// TIA Portal project "Simulador_De_Tren" (V19)

(* hardware
DEVICE "S7-1500/ET200MP station_1"  S7-1500 station
   slot 0: "Rail_0"  Rack  6ES7 590-1***0-0AA0
   slot 1: "PLC_1"  CPU 1511-1 PN  6ES7 511-1AK01-0AB0  V2.9
      slot 3: "CPU display_1"  6ES7591-1AA00-0AA0
      slot 32768: "PROFINET interface_1"  X1
         slot 32769: "Port_1"  X1 P1
         slot 32770: "Port_2"  X1 P2
      slot 34817: "Virtual CP interface port_1"  Virtual CP interface port  Virtual CP interface port
   slot 2: "DI 32x24VDC BA_1"  DI 32x24VDC BA  6ES7 521-1BL10-0AA0  V1.1
   slot 3: "DQ 32x24VDC/0.5A BA_1"  DQ 32x24VDC/0.5A BA  6ES7 522-1BL10-0AA0  V1.1
   slot 4: "AI 16xI BA_1"  AI 16xI BA  6ES7 531-7MH00-0AB0  V1.0
   slot 5: "AQ 8xU/I HS_1"  AQ 8xU/I HS  6ES7 532-5HF00-0AB0  V2.2
DEVICE "HMI_1"  TP1500 Comfort
   slot 0: "HMI_1"  TP1500 Comfort  6AV2 124-0QC02-0AX1  17.0.0.0
   slot 1: "HMI_RT_1"  TP1500 Comfort  6AV2 124-0QC02-0AX1  17.0.0.0
   slot 5: "HMI_1.IE_CP_1"  PROFINET Interface  17.0.0.0
      slot 1: "PROFINET Interface_1"  PROFINET Interface
         slot 1: "Port_1"  Port
         slot 2: "Port_2"  Port
   slot 6: "HMI_1.IE_CP_2"  PROFINET Interface  17.0.0.0
      slot 1: "PROFINET Interface_GBit"  PROFINET Interface
         slot 1: "Port_1"  Port
   slot 7: "HMI_1.MPI/DP_CP_1"  MPI/DP Interface  17.0.0.0
*)

// ===== PLC "PLC_1"  CPU 1511-1 PN =====

VAR_GLOBAL   // PLC tag table "Default tag table"
   "VT-01_TrainVibration" AT %IW4 : Int;
   "M-01-SPD_Mtr1Speed" AT %QW4 : Int;
END_VAR

VAR_GLOBAL   // PLC tag table "DigitalInputs"
   "ZS-01_LowLevel" AT %I0.0 : Bool;
   "ZS-02_HighLeve" AT %I0.1 : Bool;
   "ZS-03_MediumLevel" AT %I0.2 : Bool;
   "ZS-04" AT %I0.3 : Bool;
   "ZS-05" AT %I0.4 : Bool;
   "ZS-06" AT %I0.5 : Bool;
   "ZS-07" AT %I0.6 : Bool;
   "ZS-08" AT %I0.7 : Bool;
END_VAR

VAR_GLOBAL   // PLC tag table "DigitalOutputs"
   "M-01-Run_Mtr1RunCmd" AT %Q0.0 : Bool;
END_VAR

DATA_BLOCK "M-01"   // DB7
{ S7_Optimized_Access := 'TRUE' }
VERSION : 0.1
// stored: InstanceOfName FB_Motor_VSD
"FB_Motor_VSD"
BEGIN
END_DATA_BLOCK

DATA_BLOCK "M-02"   // DB8
{ S7_Optimized_Access := 'TRUE' }
VERSION : 0.1
// stored: InstanceOfName FB_Motor_VSD
"FB_Motor_VSD"
BEGIN
END_DATA_BLOCK

// folder: 1.IO_DB's

DATA_BLOCK "DI"   // DB1
{ S7_Optimized_Access := 'TRUE' }
VERSION : 0.1
   VAR
      "ZS-01_Fault_Rev" : Bool;
      "ZS-02_Stop1" : Bool;
      "ZS-03_Slow1_Rev" : Bool;
      "ZS-04_Slow2_Fwd" : Bool;
      "ZS-05_Stop2" : Bool;
      "ZS-06_Slow2_Rev" : Bool;
      "ZS-07_Slow3_Fwd" : Bool;
      "ZS-08_Stop3" : Bool;
      "ZS-09_Slow3_Rev" : Bool;
      "ZS-10_Slow4_Fwd" : Bool;
      "ZS-11_Stop4" : Bool;
      "ZS-12_Fault_Fwd" : Bool;
      "!XS--01_E-Stop" : Bool;
      "!XS-02_Safety_Key" : Bool;
      "!LS-01_LIght_Curtain" : Bool;
      "M-01-Ctrl_Flt" : Bool;
      "M-01-VSD_Flt" : Bool;
      "ZS-13_Brake_Engaged" : Bool;
      "M-01-Run_Conf" : Bool;
   END_VAR
BEGIN
END_DATA_BLOCK

DATA_BLOCK "DO"   // DB2
{ S7_Optimized_Access := 'TRUE' }
VERSION : 0.1
   VAR
      "XZ-01_Brake_Cmd" : Bool;
      "M-01_Run_Cmd" : Bool;
      "M-01_Mtr_Dir_Fwd" : Bool;
   END_VAR
BEGIN
END_DATA_BLOCK

DATA_BLOCK "AI"   // DB3
{ S7_Optimized_Access := 'TRUE' }
VERSION : 0.1
   VAR
      "VT-01_Train_Vibration" : Int;
   END_VAR
BEGIN
END_DATA_BLOCK

DATA_BLOCK "AO"   // DB4
{ S7_Optimized_Access := 'TRUE' }
VERSION : 0.1
   VAR
      "M-01_Mtr_Spd" : Int;
      "M-01_Mtr_Accl" : Int;
   END_VAR
BEGIN
END_DATA_BLOCK

DATA_BLOCK "HMI_Inputs"   // DB5
{ S7_Optimized_Access := 'TRUE' }
VERSION : 0.1
   VAR
      GoTo_Station1 : Bool;
      GoTo_Station2 : Bool;
      GoTo_Station3 : Bool;
      GoTo_Station4 : Bool;
   END_VAR
BEGIN
END_DATA_BLOCK

DATA_BLOCK "Const&SP"   // DB6
{ S7_Optimized_Access := 'TRUE' }
VERSION : 0.1
BEGIN
END_DATA_BLOCK

DATA_BLOCK "TestDB"   // DB9
{ S7_Optimized_Access := 'TRUE' }
VERSION : 0.1
   VAR
      Test_faultVSD : Bool;
      Test_Start : Bool;
      Test_Stop : Bool;
      Test_FWD : Bool;
      Test_Reset : Bool;
   END_VAR
BEGIN
END_DATA_BLOCK

// folder: (top level)

ORGANIZATION_BLOCK "Main"   // OB1, LAD, ProgramCycle
TITLE = "Main Program Sweep (Cycle)"
{ S7_Optimized_Access := 'TRUE' }
VERSION : 0.1
   VAR_INPUT
      Initial_Call : Bool;   // Initial call of this OB
      Remanence : Bool;   // =True, if remanent data are available
   END_VAR
BEGIN

REGION Network 1
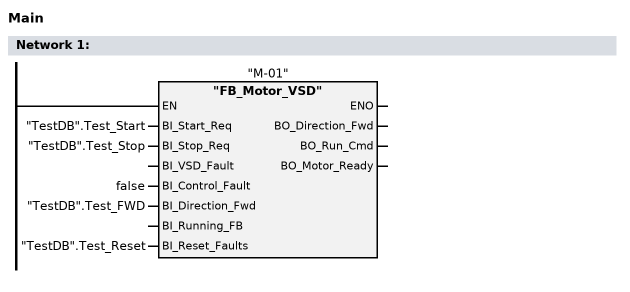
   RUNG wire#powerrail
      "M-01"(BI_Start_Req := "TestDB".Test_Start, BI_Stop_Req := "TestDB".Test_Stop, BI_VSD_Fault :=, BI_Control_Fault := false, BI_Direction_Fwd := "TestDB".Test_FWD, BI_Running_FB :=, BI_Reset_Faults := "TestDB".Test_Reset, BO_Direction_Fwd =>, BO_Run_Cmd =>, BO_Motor_Ready =>)
   END_RUNG
   // the same network as SCL:
   "M-01"(BI_Start_Req := "TestDB".Test_Start,   // "FB_Motor_VSD"
          BI_Stop_Req := "TestDB".Test_Stop,
          BI_Control_Fault := false,
          BI_Direction_Fwd := "TestDB".Test_FWD,
          BI_Reset_Faults := "TestDB".Test_Reset);
END_REGION
END_ORGANIZATION_BLOCK

// folder: 2.Function_Blocks

FUNCTION_BLOCK "FB_Motor_VSD"   // FB1, LAD
TITLE = Function block for control of a VSD Motor
{ S7_Optimized_Access := 'TRUE' }
VERSION : 0.1
   VAR_INPUT
      BI_Start_Req : Bool;
      BI_Stop_Req : Bool;
      BI_VSD_Fault : Bool;
      BI_Control_Fault : Bool;
      BI_Direction_Fwd : Bool;
      BI_Running_FB : Bool;
      BI_Reset_Faults : Bool;
   END_VAR
   VAR_OUTPUT
      BO_Direction_Fwd : Bool;
      BO_Run_Cmd : Bool;
      BO_Motor_Ready : Bool;
      BO_Running_Sts : Bool;
   END_VAR
BEGIN

REGION Network 1: Start & Stop Requests
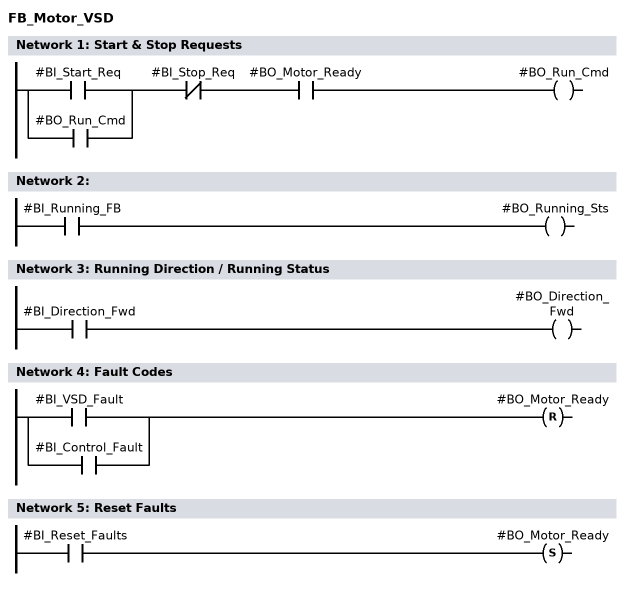
   RUNG wire#powerrail
      Contact( #BI_Start_Req )
      wire#w1
      I_Contact( #BI_Stop_Req )
      Contact( #BO_Motor_Ready )
      Coil( #BO_Run_Cmd )
   END_RUNG
   RUNG wire#powerrail
      Contact( #BO_Run_Cmd )
   END_RUNG wire#w1
   // the same network as SCL:
   #BO_Run_Cmd := (#BI_Start_Req OR #BO_Run_Cmd) AND NOT #BI_Stop_Req AND #BO_Motor_Ready;
END_REGION

REGION Network 2
   RUNG wire#powerrail
      Contact( #BI_Running_FB )
      Coil( #BO_Running_Sts )
   END_RUNG
   // the same network as SCL:
   #BO_Running_Sts := #BI_Running_FB;
END_REGION

REGION Network 3: Running Direction / Running Status
   RUNG wire#powerrail
      Contact( #BI_Direction_Fwd )
      Coil( #BO_Direction_Fwd )
   END_RUNG
   // the same network as SCL:
   #BO_Direction_Fwd := #BI_Direction_Fwd;
END_REGION

REGION Network 4: Fault Codes
   RUNG wire#powerrail
      Contact( #BI_VSD_Fault )
      wire#w1
      R_Coil( #BO_Motor_Ready )
   END_RUNG
   RUNG wire#powerrail
      Contact( #BI_Control_Fault )
   END_RUNG wire#w1
   // the same network as SCL:
   IF #BI_VSD_Fault OR #BI_Control_Fault THEN #BO_Motor_Ready := FALSE; END_IF;
END_REGION

REGION Network 5: Reset Faults
   RUNG wire#powerrail
      Contact( #BI_Reset_Faults )
      S_Coil( #BO_Motor_Ready )
   END_RUNG
   // the same network as SCL:
   IF #BI_Reset_Faults THEN #BO_Motor_Ready := TRUE; END_IF;
END_REGION
END_FUNCTION_BLOCK